    movel([0.086559, -1.204193, -2.674556, -0.833640, 1.570796, 1.657355],accel_mss,speed_ms,0,blend_radius_m)
    movel([0.088424, -1.203455, -2.674910, -0.834023, 1.570796, 1.659221],accel_mss,speed_ms,0,blend_radius_m)
    movel([0.086559, -1.204193, -2.674556, -0.833640, 1.570796, 1.657355],accel_mss,speed_ms,0,blend_radius_m)
    movel([0.088424, -1.203455, -2.674910, -0.834023, 1.570796, 1.659221],accel_mss,speed_ms,0,blend_radius_m)
    movel([0.086559, -1.204193, -2.674556, -0.833640, 1.570796, 1.657355],accel_mss,speed_ms,0,blend_radius_m)
    movel([0.086559, -1.180588, -2.662463, -0.869339, 1.570796, 1.657355],accel_mss,speed_ms,0,blend_radius_m)
    movel([0.089349, -1.179472, -2.662982, -0.869935, 1.570796, 1.660145],accel_mss,speed_ms,0,blend_radius_m)
    movel([0.089349, -1.203086, -2.675087, -0.834215, 1.570796, 1.660145],accel_mss,speed_ms,0,blend_radius_m)
    movel([0.095344, -1.200734, -2.676213, -0.835442, 1.570796, 1.666140],accel_mss,speed_ms,0,blend_radius_m)
    movel([0.089349, -1.203086, -2.675087, -0.834215, 1.570796, 1.660145],accel_mss,speed_ms,0,blend_radius_m)
    movel([0.095344, -1.200734, -2.676213, -0.835442, 1.570796, 1.666140],accel_mss,speed_ms,0,blend_radius_m)
    movel([0.089349, -1.203086, -2.675087, -0.834215, 1.570796, 1.660145],accel_mss,speed_ms,0,blend_radius_m)
    movel([0.089349, -1.179472, -2.662982, -0.869935, 1.570796, 1.660145],accel_mss,speed_ms,0,blend_radius_m)
    movel([0.098168, -1.175997, -2.664591, -0.871801, 1.570796, 1.668965],accel_mss,speed_ms,0,blend_radius_m)
    movel([0.098168, -1.199637, -2.676736, -0.836017, 1.570796, 1.668965],accel_mss,speed_ms,0,blend_radius_m)
    movel([0.107877, -1.195883, -2.678514, -0.837992, 1.570796, 1.678674],accel_mss,speed_ms,0,blend_radius_m)
    movel([0.108983, -1.195732, -2.678585, -0.838072, 1.570796, 1.679780],accel_mss,speed_ms,0,blend_radius_m)
    movel([0.109597, -1.196503, -2.678222, -0.837665, 1.570796, 1.680393],accel_mss,speed_ms,0,blend_radius_m)
    movel([0.108595, -1.204917, -2.674207, -0.833264, 1.570796, 1.679392],accel_mss,speed_ms,0,blend_radius_m)
    movel([0.106737, -1.205610, -2.673873, -0.832906, 1.570796, 1.677534],accel_mss,speed_ms,0,blend_radius_m)
    movel([0.107721, -1.197211, -2.677887, -0.837292, 1.570796, 1.678518],accel_mss,speed_ms,0,blend_radius_m)
    movel([0.098032, -1.200904, -2.676131, -0.835353, 1.570796, 1.668828],accel_mss,speed_ms,0,blend_radius_m)
    movel([0.098168, -1.199637, -2.676736, -0.836017, 1.570796, 1.668965],accel_mss,speed_ms,0,blend_radius_m)
    movel([0.107877, -1.195883, -2.678514, -0.837992, 1.570796, 1.678674],accel_mss,speed_ms,0,blend_radius_m)
    movel([0.108983, -1.195732, -2.678585, -0.838072, 1.570796, 1.679780],accel_mss,speed_ms,0,blend_radius_m)
    movel([0.109597, -1.196503, -2.678222, -0.837665, 1.570796, 1.680393],accel_mss,speed_ms,0,blend_radius_m)
    movel([0.108595, -1.204917, -2.674207, -0.833264, 1.570796, 1.679392],accel_mss,speed_ms,0,blend_radius_m)
    movel([0.106737, -1.205610, -2.673873, -0.832906, 1.570796, 1.677534],accel_mss,speed_ms,0,blend_radius_m)
    movel([0.107721, -1.197211, -2.677887, -0.837292, 1.570796, 1.678518],accel_mss,speed_ms,0,blend_radius_m)
    movel([0.098032, -1.200904, -2.676131, -0.835353, 1.570796, 1.668828],accel_mss,speed_ms,0,blend_radius_m)
    movel([0.098168, -1.199637, -2.676736, -0.836017, 1.570796, 1.668965],accel_mss,speed_ms,0,blend_radius_m)
    movel([0.098168, -1.175997, -2.664591, -0.871801, 1.570796, 1.668965],accel_mss,speed_ms,0,blend_radius_m)
    movel([0.113144, -1.170200, -2.667247, -0.874941, 1.570796, 1.683940],accel_mss,speed_ms,0,blend_radius_m)
    movel([0.113144, -1.193881, -2.679456, -0.839051, 1.570796, 1.683940],accel_mss,speed_ms,0,blend_radius_m)
    movel([0.115437, -1.193007, -2.679867, -0.839516, 1.570796, 1.686233],accel_mss,speed_ms,0,blend_radius_m)
    movel([0.117722, -1.197209, -2.677887, -0.837292, 1.570796, 1.688518],accel_mss,speed_ms,0,blend_radius_m)
    movel([0.128361, -1.193317, -2.679721, -0.839351, 1.570796, 1.699157],accel_mss,speed_ms,0,blend_radius_m)
    movel([0.129113, -1.187897, -2.682247, -0.842245, 1.570796, 1.699909],accel_mss,speed_ms,0,blend_radius_m)
    movel([0.132206, -1.186755, -2.682775, -0.842859, 1.570796, 1.703002],accel_mss,speed_ms,0,blend_radius_m)
    movel([0.131112, -1.194470, -2.679180, -0.838740, 1.570796, 1.701908],accel_mss,speed_ms,0,blend_radius_m)
    movel([0.116675, -1.199724, -2.676694, -0.835971, 1.570796, 1.687472],accel_mss,speed_ms,0,blend_radius_m)
    movel([0.115166, -1.200646, -2.676255, -0.835488, 1.570796, 1.685963],accel_mss,speed_ms,0,blend_radius_m)
    movel([0.114515, -1.201312, -2.675936, -0.835140, 1.570796, 1.685311],accel_mss,speed_ms,0,blend_radius_m)
    movel([0.113820, -1.202396, -2.675418, -0.834575, 1.570796, 1.684616],accel_mss,speed_ms,0,blend_radius_m)
    movel([0.113536, -1.203358, -2.674957, -0.834074, 1.570796, 1.684333],accel_mss,speed_ms,0,blend_radius_m)
    movel([0.113616, -1.204244, -2.674531, -0.833614, 1.570796, 1.684412],accel_mss,speed_ms,0,blend_radius_m)
    movel([0.114083, -1.204844, -2.674243, -0.833303, 1.570796, 1.684879],accel_mss,speed_ms,0,blend_radius_m)
    movel([0.114895, -1.205104, -2.674117, -0.833167, 1.570796, 1.685692],accel_mss,speed_ms,0,blend_radius_m)
    movel([0.116018, -1.204912, -2.674210, -0.833267, 1.570796, 1.686815],accel_mss,speed_ms,0,blend_radius_m)
    movel([0.130370, -1.199728, -2.676692, -0.835969, 1.570796, 1.701166],accel_mss,speed_ms,0,blend_radius_m)
    movel([0.128342, -1.202575, -2.675332, -0.834481, 1.570796, 1.699138],accel_mss,speed_ms,0,blend_radius_m)
    movel([0.116391, -1.206882, -2.673259, -0.832248, 1.570796, 1.687188],accel_mss,speed_ms,0,blend_radius_m)
    movel([0.113809, -1.207177, -2.673116, -0.832096, 1.570796, 1.684606],accel_mss,speed_ms,0,blend_radius_m)
    movel([0.112543, -1.206557, -2.673416, -0.832416, 1.570796, 1.683339],accel_mss,speed_ms,0,blend_radius_m)
    movel([0.111881, -1.205466, -2.673943, -0.832980, 1.570796, 1.682677],accel_mss,speed_ms,0,blend_radius_m)
    movel([0.111788, -1.204004, -2.674647, -0.833738, 1.570796, 1.682585],accel_mss,speed_ms,0,blend_radius_m)
    movel([0.112216, -1.202452, -2.675392, -0.834546, 1.570796, 1.683013],accel_mss,speed_ms,0,blend_radius_m)
    movel([0.113265, -1.200628, -2.676263, -0.835498, 1.570796, 1.684061],accel_mss,speed_ms,0,blend_radius_m)
    movel([0.114304, -1.199428, -2.676835, -0.836126, 1.570796, 1.685100],accel_mss,speed_ms,0,blend_radius_m)
    movel([0.115587, -1.198342, -2.677351, -0.836696, 1.570796, 1.686384],accel_mss,speed_ms,0,blend_radius_m)
    movel([0.113144, -1.193881, -2.679456, -0.839051, 1.570796, 1.683940],accel_mss,speed_ms,0,blend_radius_m)
    movel([0.115437, -1.193007, -2.679867, -0.839516, 1.570796, 1.686233],accel_mss,speed_ms,0,blend_radius_m)
    movel([0.117722, -1.197209, -2.677887, -0.837292, 1.570796, 1.688518],accel_mss,speed_ms,0,blend_radius_m)
    movel([0.128361, -1.193317, -2.679721, -0.839351, 1.570796, 1.699157],accel_mss,speed_ms,0,blend_radius_m)
    movel([0.129113, -1.187897, -2.682247, -0.842245, 1.570796, 1.699909],accel_mss,speed_ms,0,blend_radius_m)
    movel([0.132206, -1.186755, -2.682775, -0.842859, 1.570796, 1.703002],accel_mss,speed_ms,0,blend_radius_m)
    movel([0.131112, -1.194470, -2.679180, -0.838740, 1.570796, 1.701908],accel_mss,speed_ms,0,blend_radius_m)
    movel([0.116675, -1.199724, -2.676694, -0.835971, 1.570796, 1.687472],accel_mss,speed_ms,0,blend_radius_m)
    movel([0.115166, -1.200646, -2.676255, -0.835488, 1.570796, 1.685963],accel_mss,speed_ms,0,blend_radius_m)
    movel([0.114515, -1.201312, -2.675936, -0.835140, 1.570796, 1.685311],accel_mss,speed_ms,0,blend_radius_m)
    movel([0.113820, -1.202396, -2.675418, -0.834575, 1.570796, 1.684616],accel_mss,speed_ms,0,blend_radius_m)
    movel([0.113536, -1.203358, -2.674957, -0.834074, 1.570796, 1.684333],accel_mss,speed_ms,0,blend_radius_m)
    movel([0.113616, -1.204244, -2.674531, -0.833614, 1.570796, 1.684412],accel_mss,speed_ms,0,blend_radius_m)
    movel([0.114083, -1.204844, -2.674243, -0.833303, 1.570796, 1.684879],accel_mss,speed_ms,0,blend_radius_m)
    movel([0.114895, -1.205104, -2.674117, -0.833167, 1.570796, 1.685692],accel_mss,speed_ms,0,blend_radius_m)
    movel([0.116018, -1.204912, -2.674210, -0.833267, 1.570796, 1.686815],accel_mss,speed_ms,0,blend_radius_m)
    movel([0.130370, -1.199728, -2.676692, -0.835969, 1.570796, 1.701166],accel_mss,speed_ms,0,blend_radius_m)
    movel([0.128342, -1.202575, -2.675332, -0.834481, 1.570796, 1.699138],accel_mss,speed_ms,0,blend_radius_m)
    movel([0.116391, -1.206882, -2.673259, -0.832248, 1.570796, 1.687188],accel_mss,speed_ms,0,blend_radius_m)
    movel([0.113809, -1.207177, -2.673116, -0.832096, 1.570796, 1.684606],accel_mss,speed_ms,0,blend_radius_m)
    movel([0.112543, -1.206557, -2.673416, -0.832416, 1.570796, 1.683339],accel_mss,speed_ms,0,blend_radius_m)
    movel([0.111881, -1.205466, -2.673943, -0.832980, 1.570796, 1.682677],accel_mss,speed_ms,0,blend_radius_m)
    movel([0.111788, -1.204004, -2.674647, -0.833738, 1.570796, 1.682585],accel_mss,speed_ms,0,blend_radius_m)
    movel([0.112216, -1.202452, -2.675392, -0.834546, 1.570796, 1.683013],accel_mss,speed_ms,0,blend_radius_m)
    movel([0.113265, -1.200628, -2.676263, -0.835498, 1.570796, 1.684061],accel_mss,speed_ms,0,blend_radius_m)
    movel([0.114304, -1.199428, -2.676835, -0.836126, 1.570796, 1.685100],accel_mss,speed_ms,0,blend_radius_m)
    movel([0.115587, -1.198342, -2.677351, -0.836696, 1.570796, 1.686384],accel_mss,speed_ms,0,blend_radius_m)
    movel([0.113144, -1.193881, -2.679456, -0.839051, 1.570796, 1.683940],accel_mss,speed_ms,0,blend_radius_m)
    movel([0.113144, -1.170200, -2.667247, -0.874941, 1.570796, 1.683940],accel_mss,speed_ms,0,blend_radius_m)
    movel([0.134582, -1.162151, -2.670878, -0.879360, 1.570796, 1.705378],accel_mss,speed_ms,0,blend_radius_m)
    movel([0.134582, -1.185886, -2.683176, -0.843327, 1.570796, 1.705378],accel_mss,speed_ms,0,blend_radius_m)
    movel([0.137680, -1.184753, -2.683698, -0.843938, 1.570796, 1.708476],accel_mss,speed_ms,0,blend_radius_m)
    movel([0.135432, -1.200064, -2.676532, -0.835793, 1.570796, 1.706228],accel_mss,speed_ms,0,blend_radius_m)
    movel([0.132389, -1.201138, -2.676020, -0.835231, 1.570796, 1.703185],accel_mss,speed_ms,0,blend_radius_m)
    movel([0.134582, -1.185886, -2.683176, -0.843327, 1.570796, 1.705378],accel_mss,speed_ms,0,blend_radius_m)
    movel([0.137680, -1.184753, -2.683698, -0.843938, 1.570796, 1.708476],accel_mss,speed_ms,0,blend_radius_m)
    movel([0.135432, -1.200064, -2.676532, -0.835793, 1.570796, 1.706228],accel_mss,speed_ms,0,blend_radius_m)
    movel([0.132389, -1.201138, -2.676020, -0.835231, 1.570796, 1.703185],accel_mss,speed_ms,0,blend_radius_m)
    movel([0.134582, -1.185886, -2.683176, -0.843327, 1.570796, 1.705378],accel_mss,speed_ms,0,blend_radius_m)
    movel([0.134582, -1.162151, -2.670878, -0.879360, 1.570796, 1.705378],accel_mss,speed_ms,0,blend_radius_m)
    movel([0.160381, -1.152872, -2.674981, -0.884536, 1.570796, 1.731178],accel_mss,speed_ms,0,blend_radius_m)
    movel([0.160381, -1.176663, -2.687382, -0.848344, 1.570796, 1.731178],accel_mss,speed_ms,0,blend_radius_m)
    movel([0.163651, -1.175524, -2.687895, -0.848970, 1.570796, 1.734447],accel_mss,speed_ms,0,blend_radius_m)
    movel([0.149227, -1.195273, -2.678802, -0.838314, 1.570796, 1.720024],accel_mss,speed_ms,0,blend_radius_m)
    movel([0.146035, -1.196370, -2.678284, -0.837735, 1.570796, 1.716832],accel_mss,speed_ms,0,blend_radius_m)
    movel([0.139954, -1.183929, -2.684076, -0.844384, 1.570796, 1.710750],accel_mss,speed_ms,0,blend_radius_m)
    movel([0.156594, -1.177989, -2.686783, -0.847617, 1.570796, 1.727391],accel_mss,speed_ms,0,blend_radius_m)
    movel([0.139954, -1.183929, -2.684076, -0.844384, 1.570796, 1.710750],accel_mss,speed_ms,0,blend_radius_m)
    movel([0.146035, -1.196370, -2.678284, -0.837735, 1.570796, 1.716832],accel_mss,speed_ms,0,blend_radius_m)
    movel([0.149227, -1.195273, -2.678802, -0.838314, 1.570796, 1.720024],accel_mss,speed_ms,0,blend_radius_m)
    movel([0.163651, -1.175524, -2.687895, -0.848970, 1.570796, 1.734447],accel_mss,speed_ms,0,blend_radius_m)
    movel([0.160381, -1.176663, -2.687382, -0.848344, 1.570796, 1.731178],accel_mss,speed_ms,0,blend_radius_m)
    movel([0.160381, -1.152872, -2.674981, -0.884536, 1.570796, 1.731178],accel_mss,speed_ms,0,blend_radius_m)
    movel([0.160402, -1.176640, -2.687392, -0.848356, 1.570796, 1.731198],accel_mss,speed_ms,0,blend_radius_m)
    movel([0.148556, -1.192905, -2.679914, -0.839570, 1.570796, 1.719353],accel_mss,speed_ms,0,blend_radius_m)
    movel([0.144462, -1.184410, -2.683855, -0.844124, 1.570796, 1.715258],accel_mss,speed_ms,0,blend_radius_m)
    movel([0.154488, -1.180895, -2.685463, -0.846031, 1.570796, 1.725284],accel_mss,speed_ms,0,blend_radius_m)
    movel([0.156626, -1.177946, -2.686802, -0.847641, 1.570796, 1.727423],accel_mss,speed_ms,0,blend_radius_m)
    movel([0.154488, -1.180895, -2.685463, -0.846031, 1.570796, 1.725284],accel_mss,speed_ms,0,blend_radius_m)
    movel([0.144462, -1.184410, -2.683855, -0.844124, 1.570796, 1.715258],accel_mss,speed_ms,0,blend_radius_m)
    movel([0.148556, -1.192905, -2.679914, -0.839570, 1.570796, 1.719353],accel_mss,speed_ms,0,blend_radius_m)
    movel([0.160402, -1.176640, -2.687392, -0.848356, 1.570796, 1.731198],accel_mss,speed_ms,0,blend_radius_m)
    movel([0.160402, -1.152849, -2.674991, -0.884549, 1.570796, 1.731198],accel_mss,speed_ms,0,blend_radius_m)
    movel([0.127960, -1.169778, -2.667440, -0.875172, 1.570796, 1.698757],accel_mss,speed_ms,0,blend_radius_m)
    movel([0.127960, -1.193462, -2.679653, -0.839274, 1.570796, 1.698757],accel_mss,speed_ms,0,blend_radius_m)
    movel([0.117722, -1.197209, -2.677887, -0.837292, 1.570796, 1.688518],accel_mss,speed_ms,0,blend_radius_m)
    movel([0.127960, -1.193462, -2.679653, -0.839274, 1.570796, 1.698757],accel_mss,speed_ms,0,blend_radius_m)
    movel([0.127960, -1.169778, -2.667440, -0.875172, 1.570796, 1.698757],accel_mss,speed_ms,0,blend_radius_m)
    movel([0.126927, -1.177330, -2.663976, -0.871084, 1.570796, 1.697724],accel_mss,speed_ms,0,blend_radius_m)
    movel([0.126927, -1.200959, -2.676105, -0.835324, 1.570796, 1.697724],accel_mss,speed_ms,0,blend_radius_m)
    movel([0.116018, -1.204912, -2.674210, -0.833267, 1.570796, 1.686815],accel_mss,speed_ms,0,blend_radius_m)
    movel([0.126927, -1.200959, -2.676105, -0.835324, 1.570796, 1.697724],accel_mss,speed_ms,0,blend_radius_m)
    movel([0.126927, -1.177330, -2.663976, -0.871084, 1.570796, 1.697724],accel_mss,speed_ms,0,blend_radius_m)
    movel([0.128342, -1.178957, -2.663221, -0.870211, 1.570796, 1.699138],accel_mss,speed_ms,0,blend_radius_m)
    movel([0.128342, -1.202575, -2.675332, -0.834481, 1.570796, 1.699138],accel_mss,speed_ms,0,blend_radius_m)
    movel([0.116391, -1.206882, -2.673259, -0.832248, 1.570796, 1.687188],accel_mss,speed_ms,0,blend_radius_m)
    movel([0.128342, -1.202575, -2.675332, -0.834481, 1.570796, 1.699138],accel_mss,speed_ms,0,blend_radius_m)
    movel([0.128342, -1.178957, -2.663221, -0.870211, 1.570796, 1.699138],accel_mss,speed_ms,0,blend_radius_m)
    movel([0.087681, -1.187374, -2.659275, -0.865740, 1.570796, 1.658478],accel_mss,speed_ms,0,blend_radius_m)
    movel([0.087681, -1.210927, -2.671293, -0.830170, 1.570796, 1.658478],accel_mss,speed_ms,0,blend_radius_m)
    movel([0.094556, -1.208282, -2.672580, -0.831527, 1.570796, 1.665352],accel_mss,speed_ms,0,blend_radius_m)
    movel([0.087681, -1.210927, -2.671293, -0.830170, 1.570796, 1.658478],accel_mss,speed_ms,0,blend_radius_m)
    movel([0.094556, -1.208282, -2.672580, -0.831527, 1.570796, 1.665352],accel_mss,speed_ms,0,blend_radius_m)
    movel([0.087681, -1.210927, -2.671293, -0.830170, 1.570796, 1.658478],accel_mss,speed_ms,0,blend_radius_m)
    movel([0.087681, -1.187374, -2.659275, -0.865740, 1.570796, 1.658478],accel_mss,speed_ms,0,blend_radius_m)
    movel([0.080158, -1.190327, -2.657873, -0.864189, 1.570796, 1.650954],accel_mss,speed_ms,0,blend_radius_m)
    movel([0.080158, -1.213855, -2.669858, -0.828677, 1.570796, 1.650954],accel_mss,speed_ms,0,blend_radius_m)
    movel([0.074120, -1.216230, -2.668686, -0.827472, 1.570796, 1.644916],accel_mss,speed_ms,0,blend_radius_m)
    movel([0.080158, -1.213855, -2.669858, -0.828677, 1.570796, 1.650954],accel_mss,speed_ms,0,blend_radius_m)
    movel([0.080158, -1.190327, -2.657873, -0.864189, 1.570796, 1.650954],accel_mss,speed_ms,0,blend_radius_m)
    movel([0.095344, -1.177102, -2.664081, -0.871206, 1.570796, 1.666140],accel_mss,speed_ms,0,blend_radius_m)
    movel([0.095344, -1.200734, -2.676213, -0.835442, 1.570796, 1.666140],accel_mss,speed_ms,0,blend_radius_m)
    movel([0.096311, -1.200542, -2.676304, -0.835542, 1.570796, 1.667107],accel_mss,speed_ms,0,blend_radius_m)
    movel([0.097080, -1.201270, -2.675957, -0.835162, 1.570796, 1.667877],accel_mss,speed_ms,0,blend_radius_m)
    movel([0.096543, -1.206327, -2.673527, -0.832535, 1.570796, 1.667339],accel_mss,speed_ms,0,blend_radius_m)
    movel([0.097080, -1.201270, -2.675957, -0.835162, 1.570796, 1.667877],accel_mss,speed_ms,0,blend_radius_m)
    movel([0.096311, -1.200542, -2.676304, -0.835542, 1.570796, 1.667107],accel_mss,speed_ms,0,blend_radius_m)
    movel([0.095344, -1.200734, -2.676213, -0.835442, 1.570796, 1.666140],accel_mss,speed_ms,0,blend_radius_m)
    movel([0.095344, -1.177102, -2.664081, -0.871206, 1.570796, 1.666140],accel_mss,speed_ms,0,blend_radius_m)
    movel([0.089349, -1.179472, -2.662982, -0.869935, 1.570796, 1.660145],accel_mss,speed_ms,0,blend_radius_m)
    movel([0.089349, -1.203086, -2.675087, -0.834215, 1.570796, 1.660145],accel_mss,speed_ms,0,blend_radius_m)
    movel([0.089229, -1.204311, -2.674499, -0.833579, 1.570796, 1.660025],accel_mss,speed_ms,0,blend_radius_m)
    movel([0.095213, -1.201990, -2.675613, -0.834786, 1.570796, 1.666009],accel_mss,speed_ms,0,blend_radius_m)
    movel([0.094686, -1.207038, -2.673183, -0.832168, 1.570796, 1.665482],accel_mss,speed_ms,0,blend_radius_m)
    movel([0.087815, -1.209715, -2.671883, -0.830790, 1.570796, 1.658612],accel_mss,speed_ms,0,blend_radius_m)
    movel([0.088424, -1.203455, -2.674910, -0.834023, 1.570796, 1.659221],accel_mss,speed_ms,0,blend_radius_m)
    movel([0.087815, -1.209715, -2.671883, -0.830790, 1.570796, 1.658612],accel_mss,speed_ms,0,blend_radius_m)
    movel([0.094686, -1.207038, -2.673183, -0.832168, 1.570796, 1.665482],accel_mss,speed_ms,0,blend_radius_m)
    movel([0.095213, -1.201990, -2.675613, -0.834786, 1.570796, 1.666009],accel_mss,speed_ms,0,blend_radius_m)
    movel([0.089229, -1.204311, -2.674499, -0.833579, 1.570796, 1.660025],accel_mss,speed_ms,0,blend_radius_m)
    movel([0.089349, -1.203086, -2.675087, -0.834215, 1.570796, 1.660145],accel_mss,speed_ms,0,blend_radius_m)
    movel([0.089349, -1.179472, -2.662982, -0.869935, 1.570796, 1.660145],accel_mss,speed_ms,0,blend_radius_m)
    movel([0.087699, -1.187368, -2.659278, -0.865743, 1.570796, 1.658495],accel_mss,speed_ms,0,blend_radius_m)
    movel([0.087699, -1.210920, -2.671296, -0.830173, 1.570796, 1.658495],accel_mss,speed_ms,0,blend_radius_m)
    movel([0.086535, -1.211101, -2.671207, -0.830081, 1.570796, 1.657332],accel_mss,speed_ms,0,blend_radius_m)
    movel([0.085963, -1.210442, -2.671529, -0.830418, 1.570796, 1.656760],accel_mss,speed_ms,0,blend_radius_m)
    movel([0.086559, -1.204193, -2.674556, -0.833640, 1.570796, 1.657355],accel_mss,speed_ms,0,blend_radius_m)
    movel([0.085963, -1.210442, -2.671529, -0.830418, 1.570796, 1.656760],accel_mss,speed_ms,0,blend_radius_m)
    movel([0.086535, -1.211101, -2.671207, -0.830081, 1.570796, 1.657332],accel_mss,speed_ms,0,blend_radius_m)
    movel([0.087699, -1.210920, -2.671296, -0.830173, 1.570796, 1.658495],accel_mss,speed_ms,0,blend_radius_m)
    movel([0.087699, -1.187368, -2.659278, -0.865743, 1.570796, 1.658495],accel_mss,speed_ms,0,blend_radius_m)
    movel([0.072371, -1.192322, -2.656920, -0.863147, 1.570796, 1.643167],accel_mss,speed_ms,0,blend_radius_m)
    movel([0.072371, -1.215834, -2.668882, -0.827673, 1.570796, 1.643167],accel_mss,speed_ms,0,blend_radius_m)
    movel([0.072777, -1.210807, -2.671351, -0.830231, 1.570796, 1.643574],accel_mss,speed_ms,0,blend_radius_m)
    movel([0.072371, -1.215834, -2.668882, -0.827673, 1.570796, 1.643167],accel_mss,speed_ms,0,blend_radius_m)
    movel([0.072371, -1.192322, -2.656920, -0.863147, 1.570796, 1.643167],accel_mss,speed_ms,0,blend_radius_m)
    movel([0.107877, -1.172216, -2.666328, -0.873845, 1.570796, 1.678674],accel_mss,speed_ms,0,blend_radius_m)
    movel([0.107877, -1.195883, -2.678514, -0.837992, 1.570796, 1.678674],accel_mss,speed_ms,0,blend_radius_m)
    movel([0.098168, -1.199637, -2.676736, -0.836017, 1.570796, 1.668965],accel_mss,speed_ms,0,blend_radius_m)
    movel([0.107877, -1.195883, -2.678514, -0.837992, 1.570796, 1.678674],accel_mss,speed_ms,0,blend_radius_m)
    movel([0.107877, -1.172216, -2.666328, -0.873845, 1.570796, 1.678674],accel_mss,speed_ms,0,blend_radius_m)
    movel([0.096543, -1.182730, -2.661462, -0.868197, 1.570796, 1.667340],accel_mss,speed_ms,0,blend_radius_m)
    movel([0.096543, -1.206319, -2.673531, -0.832539, 1.570796, 1.667340],accel_mss,speed_ms,0,blend_radius_m)
    movel([0.095536, -1.207734, -2.672846, -0.831809, 1.570796, 1.666333],accel_mss,speed_ms,0,blend_radius_m)
    movel([0.094556, -1.208282, -2.672580, -0.831527, 1.570796, 1.665352],accel_mss,speed_ms,0,blend_radius_m)
    movel([0.095536, -1.207734, -2.672846, -0.831809, 1.570796, 1.666333],accel_mss,speed_ms,0,blend_radius_m)
    movel([0.096543, -1.206319, -2.673531, -0.832539, 1.570796, 1.667340],accel_mss,speed_ms,0,blend_radius_m)
    movel([0.096543, -1.139938, -2.636350, -0.936101, 1.570796, 1.667340],accel_mss,speed_ms,0,blend_radius_m)
    # End of main program
  end

  Machining1()
end
